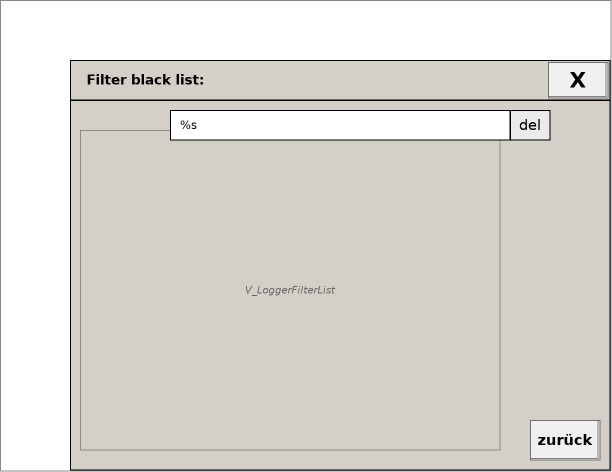
VISUALIZATION V_LoggerFilterBlack  // 612x472
    Rectangle (70,100 540x370)
    Rectangle (70,60 540x40), "Filter black list:"
    Frame (80,130 420x320)
        shows V_LoggerFilterList(IOfbLogger := gfbLogger, IOszFilterTxt := gfbLogger.szVisuFilterBlack)
    Rectangle (170,110 340x30), "%s", tooltip "whitelist: Begriff1[;Begriff2[;Begriff3]]", text variable: gfbLogger.szVisuFilterBlack
        OnMouseClick: write the text variable via Default
    Rectangle (510,110 40x30), "del", tooltip "löschen"
        OnMouseClick: execute { gfbLogger.szVisuFilterBlack := ''; }
    Button (530,420 70x40), "zurück"
        OnMouseClick: change screen: Previous 
    Button (548,62 60x36), "X"
        OnMouseClick: change screen: Previous 
END_VISUALIZATION

(* stored: Version 1.1.0.1, ProductVersion 3.1.4018.10
   Visu V_LoggerFilterBlack: Id {ecd51f36-0561-45c5-afae-4281a30419a6} *)
